Fanuc TP program (LS listing): ground_truth.ls

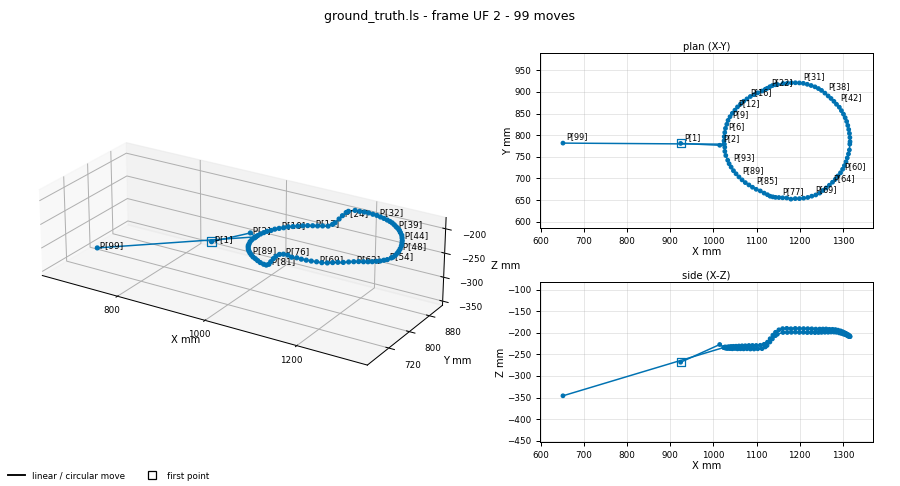
[picture p0: tool path of ground_truth.ls in frame UF 2, 99 of 99 moves have a stored position in this frame; points joined in program order, loops and branches not executed]
/PROG  TOR_XL_LEARN_V10
/ATTR
OWNER		= MNEDITOR;
COMMENT		= "WeldPRO Auto-Gen";
PROG_SIZE	= 7125;
CREATE		= DATE 26-07-31  TIME 15:22:18;
MODIFIED	= DATE 26-07-31  TIME 15:55:46;
FILE_NAME	= TOR_XL_L;
VERSION		= 0;
LINE_COUNT	= 113;
MEMORY_SIZE	= 7445;
PROTECT		= READ_WRITE;
TCD:  STACK_SIZE	= 0,
      TASK_PRIORITY	= 50,
      TIME_SLICE	= 0,
      BUSY_LAMP_OFF	= 0,
      ABORT_REQUEST	= 0,
      PAUSE_REQUEST	= 0;
DEFAULT_GROUP	= 1,*,*,*,*;
CONTROL_CODE	= 00000000 00000000;
/APPL
/MN
   1:  !WeldPRO Auto-Generated TPP ;
   2:  !TOR_XL_2026, TOR_xl_2907 ;
   3:   ;
   4:  UFRAME_NUM=2 ;
   5:  UTOOL_NUM=2 ;
   6:  !Feature Approach ;
   7:J P[1] 100% FINE    ;
   8:   ;
   9:  !Segment1 ;
  10:L P[2] 2000mm/sec FINE    ;
  11:   ;
  12:  CALL LASER_OFF    ;
  13:L P[3] R[23:moving]mm/sec CNT100    ;
  14:L P[4] R[23:moving]mm/sec CNT100    ;
  15:L P[5] R[23:moving]mm/sec CNT100    ;
  16:L P[6] R[23:moving]mm/sec CNT100    ;
  17:L P[7] R[23:moving]mm/sec CNT100    ;
  18:L P[8] R[23:moving]mm/sec CNT100    ;
  19:L P[9] R[23:moving]mm/sec CNT100    ;
  20:L P[10] R[23:moving]mm/sec CNT100    ;
  21:L P[11] R[23:moving]mm/sec CNT100    ;
  22:L P[12] R[23:moving]mm/sec CNT100    ;
  23:L P[13] R[23:moving]mm/sec CNT100    ;
  24:L P[14] R[23:moving]mm/sec CNT100    ;
  25:L P[15] R[23:moving]mm/sec CNT100    ;
  26:L P[16] R[23:moving]mm/sec CNT100    ;
  27:L P[17] R[23:moving]mm/sec CNT100    ;
  28:L P[18] R[23:moving]mm/sec CNT100    ;
  29:L P[19] R[23:moving]mm/sec CNT100    ;
  30:L P[20] R[23:moving]mm/sec CNT100    ;
  31:L P[21] R[23:moving]mm/sec CNT100    ;
  32:L P[22] R[23:moving]mm/sec CNT100    ;
  33:L P[23] R[23:moving]mm/sec CNT100    ;
  34:L P[24] R[23:moving]mm/sec CNT100    ;
  35:L P[25] R[23:moving]mm/sec CNT100    ;
  36:L P[26] R[23:moving]mm/sec CNT100    ;
  37:L P[27] R[23:moving]mm/sec CNT100    ;
  38:L P[28] R[23:moving]mm/sec CNT100    ;
  39:L P[29] R[23:moving]mm/sec CNT100    ;
  40:L P[30] R[23:moving]mm/sec CNT100    ;
  41:L P[31] R[23:moving]mm/sec CNT100    ;
  42:L P[32] R[23:moving]mm/sec CNT100    ;
  43:L P[33] R[23:moving]mm/sec CNT100    ;
  44:L P[34] R[23:moving]mm/sec CNT100    ;
  45:L P[35] R[23:moving]mm/sec CNT100    ;
  46:L P[36] R[23:moving]mm/sec CNT100    ;
  47:L P[37] R[23:moving]mm/sec CNT100    ;
  48:L P[38] R[23:moving]mm/sec CNT100    ;
  49:L P[39] R[23:moving]mm/sec CNT100    ;
  50:L P[40] R[23:moving]mm/sec CNT100    ;
  51:L P[41] R[23:moving]mm/sec CNT100    ;
  52:L P[42] R[23:moving]mm/sec CNT100    ;
  53:L P[43] R[23:moving]mm/sec CNT100    ;
  54:L P[44] R[23:moving]mm/sec CNT100    ;
  55:L P[45] R[23:moving]mm/sec CNT100    ;
  56:L P[46] R[23:moving]mm/sec CNT100    ;
  57:L P[47] R[23:moving]mm/sec CNT100    ;
  58:L P[48] R[23:moving]mm/sec CNT100    ;
  59:L P[49] R[23:moving]mm/sec CNT100    ;
  60:L P[50] R[23:moving]mm/sec CNT100    ;
  61:L P[51] R[23:moving]mm/sec CNT100    ;
  62:L P[52] R[23:moving]mm/sec CNT100    ;
  63:L P[53] R[23:moving]mm/sec CNT100    ;
  64:L P[54] R[23:moving]mm/sec CNT100    ;
  65:L P[55] R[23:moving]mm/sec CNT100    ;
  66:L P[56] R[23:moving]mm/sec CNT100    ;
  67:L P[57] R[23:moving]mm/sec CNT100    ;
  68:L P[58] R[23:moving]mm/sec CNT100    ;
  69:L P[59] R[23:moving]mm/sec CNT100    ;
  70:L P[60] R[23:moving]mm/sec CNT100    ;
  71:L P[61] R[23:moving]mm/sec CNT100    ;
  72:L P[62] R[23:moving]mm/sec CNT100    ;
  73:L P[63] R[23:moving]mm/sec CNT100    ;
  74:L P[64] R[23:moving]mm/sec CNT100    ;
  75:L P[65] R[23:moving]mm/sec CNT100    ;
  76:L P[66] R[23:moving]mm/sec CNT100    ;
  77:L P[67] R[23:moving]mm/sec CNT100    ;
  78:L P[68] R[23:moving]mm/sec CNT100    ;
  79:L P[69] R[23:moving]mm/sec CNT100    ;
  80:L P[70] R[23:moving]mm/sec CNT100    ;
  81:L P[71] R[23:moving]mm/sec CNT100    ;
  82:L P[72] R[23:moving]mm/sec CNT100    ;
  83:L P[73] R[23:moving]mm/sec CNT100    ;
  84:L P[74] R[23:moving]mm/sec CNT100    ;
  85:L P[75] R[23:moving]mm/sec CNT100    ;
  86:L P[76] R[23:moving]mm/sec CNT100    ;
  87:L P[77] R[23:moving]mm/sec CNT100    ;
  88:L P[78] R[23:moving]mm/sec CNT100    ;
  89:L P[79] R[23:moving]mm/sec CNT100    ;
  90:L P[80] R[23:moving]mm/sec CNT100    ;
  91:L P[81] R[23:moving]mm/sec CNT100    ;
  92:L P[82] R[23:moving]mm/sec CNT100    ;
  93:L P[83] R[23:moving]mm/sec CNT100    ;
  94:L P[84] R[23:moving]mm/sec CNT100    ;
  95:L P[85] R[23:moving]mm/sec CNT100    ;
  96:L P[86] R[23:moving]mm/sec CNT100    ;
  97:L P[87] R[23:moving]mm/sec CNT100    ;
  98:L P[88] R[23:moving]mm/sec CNT100    ;
  99:L P[89] R[23:moving]mm/sec CNT100    ;
 100:L P[90] R[23:moving]mm/sec CNT100    ;
 101:L P[91] R[23:moving]mm/sec CNT100    ;
 102:L P[92] R[23:moving]mm/sec CNT100    ;
 103:L P[93] R[23:moving]mm/sec CNT100    ;
 104:L P[94] R[23:moving]mm/sec CNT100    ;
 105:L P[95] R[23:moving]mm/sec CNT100    ;
 106:L P[96] R[23:moving]mm/sec CNT100    ;
 107:L P[97] R[23:moving]mm/sec CNT100    ;
 108:L P[98] R[23:moving]mm/sec FINE    ;
 109:  CALL LASER_OFF    ;
 110:   ;
 111:  !Feature Retreat ;
 112:L P[99] 2000mm/sec FINE    ;
 113:  CALL ROTATE    ;
/POS
P[1]{
   GP1:
	UF : 2, UT : 2,		CONFIG : 'F D T, 0, 0, 0',
	X =   924.335  mm,	Y =   780.986  mm,	Z =  -268.284  mm,
	W =  -106.495 deg,	P =   -15.000 deg,	R =    94.234 deg
};
P[2]{
   GP1:
	UF : 2, UT : 2,		CONFIG : 'F D T, 0, 0, 0',
	X =  1014.789  mm,	Y =   776.665  mm,	Z =  -227.278  mm,
	W =  -106.497 deg,	P =   -14.995 deg,	R =    94.216 deg
};
P[3]{
   GP1:
	UF : 2, UT : 2,		CONFIG : 'F D T, 0, 0, 0',
	X =  1024.819  mm,	Y =   779.312  mm,	Z =  -234.214  mm,
	W =  -106.501 deg,	P =   -14.998 deg,	R =    94.232 deg
};
P[4]{
   GP1:
	UF : 2, UT : 2,		CONFIG : 'F D T, 0, 0, 0',
	X =  1024.807  mm,	Y =   787.035  mm,	Z =  -234.284  mm,
	W =  -106.497 deg,	P =   -15.098 deg,	R =    90.375 deg
};
P[5]{
   GP1:
	UF : 2, UT : 2,		CONFIG : 'F D T, 0, 0, 0',
	X =  1025.197  mm,	Y =   796.630  mm,	Z =  -234.431  mm,
	W =  -106.481 deg,	P =   -15.217 deg,	R =    85.597 deg
};
P[6]{
   GP1:
	UF : 2, UT : 2,		CONFIG : 'F D T, 0, 0, 0',
	X =  1026.459  mm,	Y =   806.252  mm,	Z =  -234.929  mm,
	W =  -106.456 deg,	P =   -15.334 deg,	R =    80.807 deg
};
P[7]{
   GP1:
	UF : 2, UT : 2,		CONFIG : 'F D T, 0, 0, 0',
	X =  1028.142  mm,	Y =   815.795  mm,	Z =  -235.323  mm,
	W =  -106.423 deg,	P =   -15.450 deg,	R =    76.083 deg
};
P[8]{
   GP1:
	UF : 2, UT : 2,		CONFIG : 'F D T, 0, 0, 0',
	X =  1031.142  mm,	Y =   825.143  mm,	Z =  -236.265  mm,
	W =  -106.379 deg,	P =   -15.565 deg,	R =    71.210 deg
};
P[9]{
   GP1:
	UF : 2, UT : 2,		CONFIG : 'F D T, 0, 0, 0',
	X =  1034.075  mm,	Y =   834.282  mm,	Z =  -236.286  mm,
	W =  -106.322 deg,	P =   -15.679 deg,	R =    66.207 deg
};
P[10]{
   GP1:
	UF : 2, UT : 2,		CONFIG : 'F D T, 0, 0, 0',
	X =  1038.673  mm,	Y =   842.768  mm,	Z =  -236.720  mm,
	W =  -106.254 deg,	P =   -15.791 deg,	R =    61.015 deg
};
P[11]{
   GP1:
	UF : 2, UT : 2,		CONFIG : 'F D T, 0, 0, 0',
	X =  1044.018  mm,	Y =   850.684  mm,	Z =  -237.130  mm,
	W =  -106.180 deg,	P =   -15.896 deg,	R =    55.976 deg
};
P[12]{
   GP1:
	UF : 2, UT : 2,		CONFIG : 'F D T, 0, 0, 0',
	X =  1049.984  mm,	Y =   857.894  mm,	Z =  -236.475  mm,
	W =  -106.096 deg,	P =   -15.986 deg,	R =    51.162 deg
};
P[13]{
   GP1:
	UF : 2, UT : 2,		CONFIG : 'F D T, 0, 0, 0',
	X =  1055.988  mm,	Y =   865.483  mm,	Z =  -237.302  mm,
	W =  -106.012 deg,	P =   -16.067 deg,	R =    46.628 deg
};
P[14]{
   GP1:
	UF : 2, UT : 2,		CONFIG : 'F D T, 0, 0, 0',
	X =  1062.915  mm,	Y =   871.946  mm,	Z =  -237.205  mm,
	W =  -105.919 deg,	P =   -16.142 deg,	R =    41.952 deg
};
P[15]{
   GP1:
	UF : 2, UT : 2,		CONFIG : 'F D T, 0, 0, 0',
	X =  1070.115  mm,	Y =   878.600  mm,	Z =  -237.364  mm,
	W =  -105.870 deg,	P =   -16.177 deg,	R =    39.609 deg
};
P[16]{
   GP1:
	UF : 2, UT : 2,		CONFIG : 'F D T, 0, 0, 0',
	X =  1077.825  mm,	Y =   884.048  mm,	Z =  -237.128  mm,
	W =  -105.777 deg,	P =   -16.235 deg,	R =    35.365 deg
};
P[17]{
   GP1:
	UF : 2, UT : 2,		CONFIG : 'F D T, 0, 0, 0',
	X =  1085.741  mm,	Y =   889.534  mm,	Z =  -237.642  mm,
	W =  -105.677 deg,	P =   -16.289 deg,	R =    30.964 deg
};
P[18]{
   GP1:
	UF : 2, UT : 2,		CONFIG : 'F D T, 0, 0, 0',
	X =  1094.256  mm,	Y =   893.782  mm,	Z =  -237.649  mm,
	W =  -105.579 deg,	P =   -16.333 deg,	R =    26.830 deg
};
P[19]{
   GP1:
	UF : 2, UT : 2,		CONFIG : 'F D T, 0, 0, 0',
	X =  1102.826  mm,	Y =   898.014  mm,	Z =  -237.175  mm,
	W =  -105.535 deg,	P =   -16.344 deg,	R =    25.007 deg
};
P[20]{
   GP1:
	UF : 2, UT : 2,		CONFIG : 'F D T, 0, 0, 0',
	X =  1112.677  mm,	Y =   902.287  mm,	Z =  -236.848  mm,
	W =  -116.027 deg,	P =   -16.063 deg,	R =    30.267 deg
};
P[21]{
   GP1:
	UF : 2, UT : 2,		CONFIG : 'F D T, 0, 0, 0',
	X =  1120.220  mm,	Y =   906.262  mm,	Z =  -232.858  mm,
	W =  -126.877 deg,	P =   -15.356 deg,	R =    25.893 deg
};
P[22]{
   GP1:
	UF : 2, UT : 2,		CONFIG : 'F D T, 0, 0, 0',
	X =  1124.394  mm,	Y =   908.354  mm,	Z =  -229.385  mm,
	W =  -121.184 deg,	P =   -15.973 deg,	R =    18.444 deg
};
P[23]{
   GP1:
	UF : 2, UT : 2,		CONFIG : 'F D T, 0, 0, 0',
	X =  1130.913  mm,	Y =   912.231  mm,	Z =  -221.471  mm,
	W =  -115.329 deg,	P =   -16.208 deg,	R =    11.788 deg
};
P[24]{
   GP1:
	UF : 2, UT : 2,		CONFIG : 'F D T, 0, 0, 0',
	X =  1136.659  mm,	Y =   914.820  mm,	Z =  -214.206  mm,
	W =  -112.639 deg,	P =   -16.315 deg,	R =     9.714 deg
};
P[25]{
   GP1:
	UF : 2, UT : 2,		CONFIG : 'F D T, 0, 0, 0',
	X =  1143.585  mm,	Y =   916.753  mm,	Z =  -206.769  mm,
	W =  -110.015 deg,	P =   -16.386 deg,	R =     9.649 deg
};
P[26]{
   GP1:
	UF : 2, UT : 2,		CONFIG : 'F D T, 0, 0, 0',
	X =  1148.127  mm,	Y =   917.333  mm,	Z =  -203.429  mm,
	W =  -108.552 deg,	P =   -16.418 deg,	R =     8.950 deg
};
P[27]{
   GP1:
	UF : 2, UT : 2,		CONFIG : 'F D T, 0, 0, 0',
	X =  1161.287  mm,	Y =   919.693  mm,	Z =  -199.396  mm,
	W =  -105.409 deg,	P =   -16.443 deg,	R =     6.805 deg
};
P[28]{
   GP1:
	UF : 2, UT : 2,		CONFIG : 'F D T, 0, 0, 0',
	X =  1171.157  mm,	Y =   920.269  mm,	Z =  -199.402  mm,
	W =  -104.866 deg,	P =   -16.444 deg,	R =     5.597 deg
};
P[29]{
   GP1:
	UF : 2, UT : 2,		CONFIG : 'F D T, 0, 0, 0',
	X =  1180.649  mm,	Y =   921.254  mm,	Z =  -199.064  mm,
	W =  -104.887 deg,	P =   -16.444 deg,	R =     3.523 deg
};
P[30]{
   GP1:
	UF : 2, UT : 2,		CONFIG : 'F D T, 0, 0, 0',
	X =  1189.853  mm,	Y =   921.397  mm,	Z =  -198.761  mm,
	W =  -104.930 deg,	P =   -16.439 deg,	R =     -.729 deg
};
P[31]{
   GP1:
	UF : 2, UT : 2,		CONFIG : 'F D T, 0, 0, 0',
	X =  1199.182  mm,	Y =   920.957  mm,	Z =  -199.232  mm,
	W =  -104.979 deg,	P =   -16.424 deg,	R =    -5.541 deg
};
P[32]{
   GP1:
	UF : 2, UT : 2,		CONFIG : 'F D T, 0, 0, 0',
	X =  1208.351  mm,	Y =   920.022  mm,	Z =  -199.133  mm,
	W =  -105.028 deg,	P =   -16.400 deg,	R =   -10.259 deg
};
P[33]{
   GP1:
	UF : 2, UT : 2,		CONFIG : 'F D T, 0, 0, 0',
	X =  1217.485  mm,	Y =   917.761  mm,	Z =  -199.566  mm,
	W =  -105.070 deg,	P =   -16.371 deg,	R =   -14.490 deg
};
P[34]{
   GP1:
	UF : 2, UT : 2,		CONFIG : 'F D T, 0, 0, 0',
	X =  1226.426  mm,	Y =   915.001  mm,	Z =  -199.462  mm,
	W =  -105.112 deg,	P =   -16.334 deg,	R =   -18.515 deg
};
P[35]{
   GP1:
	UF : 2, UT : 2,		CONFIG : 'F D T, 0, 0, 0',
	X =  1235.239  mm,	Y =   911.936  mm,	Z =  -199.665  mm,
	W =  -105.158 deg,	P =   -16.285 deg,	R =   -23.051 deg
};
P[36]{
   GP1:
	UF : 2, UT : 2,		CONFIG : 'F D T, 0, 0, 0',
	X =  1243.244  mm,	Y =   907.972  mm,	Z =  -199.458  mm,
	W =  -105.219 deg,	P =   -16.204 deg,	R =   -29.417 deg
};
P[37]{
   GP1:
	UF : 2, UT : 2,		CONFIG : 'F D T, 0, 0, 0',
	X =  1250.416  mm,	Y =   903.609  mm,	Z =  -199.147  mm,
	W =  -105.311 deg,	P =   -16.047 deg,	R =   -39.415 deg
};
P[38]{
   GP1:
	UF : 2, UT : 2,		CONFIG : 'F D T, 0, 0, 0',
	X =  1258.217  mm,	Y =   897.390  mm,	Z =  -198.941  mm,
	W =  -105.307 deg,	P =   -16.055 deg,	R =   -38.974 deg
};
P[39]{
   GP1:
	UF : 2, UT : 2,		CONFIG : 'F D T, 0, 0, 0',
	X =  1265.775  mm,	Y =   890.850  mm,	Z =  -198.923  mm,
	W =  -105.302 deg,	P =   -16.063 deg,	R =   -38.625 deg
};
P[40]{
   GP1:
	UF : 2, UT : 2,		CONFIG : 'F D T, 0, 0, 0',
	X =  1272.442  mm,	Y =   885.004  mm,	Z =  -198.403  mm,
	W =  -105.469 deg,	P =   -15.944 deg,	R =   -44.977 deg
};
P[41]{
   GP1:
	UF : 2, UT : 2,		CONFIG : 'F D T, 0, 0, 0',
	X =  1279.129  mm,	Y =   878.386  mm,	Z =  -198.494  mm,
	W =  -105.661 deg,	P =   -15.890 deg,	R =   -47.714 deg
};
P[42]{
   GP1:
	UF : 2, UT : 2,		CONFIG : 'F D T, 0, 0, 0',
	X =  1285.054  mm,	Y =   871.499  mm,	Z =  -198.979  mm,
	W =  -106.210 deg,	P =   -15.792 deg,	R =   -52.259 deg
};
P[43]{
   GP1:
	UF : 2, UT : 2,		CONFIG : 'F D T, 0, 0, 0',
	X =  1291.590  mm,	Y =   864.741  mm,	Z =  -200.433  mm,
	W =  -106.927 deg,	P =   -15.688 deg,	R =   -56.663 deg
};
P[44]{
   GP1:
	UF : 2, UT : 2,		CONFIG : 'F D T, 0, 0, 0',
	X =  1296.495  mm,	Y =   856.855  mm,	Z =  -201.631  mm,
	W =  -107.603 deg,	P =   -15.597 deg,	R =   -60.244 deg
};
P[45]{
   GP1:
	UF : 2, UT : 2,		CONFIG : 'F D T, 0, 0, 0',
	X =  1301.221  mm,	Y =   848.739  mm,	Z =  -203.247  mm,
	W =  -108.271 deg,	P =   -15.504 deg,	R =   -63.686 deg
};
P[46]{
   GP1:
	UF : 2, UT : 2,		CONFIG : 'F D T, 0, 0, 0',
	X =  1305.143  mm,	Y =   840.488  mm,	Z =  -204.302  mm,
	W =  -109.143 deg,	P =   -15.378 deg,	R =   -68.203 deg
};
P[47]{
   GP1:
	UF : 2, UT : 2,		CONFIG : 'F D T, 0, 0, 0',
	X =  1308.602  mm,	Y =   831.819  mm,	Z =  -205.714  mm,
	W =  -109.899 deg,	P =   -15.253 deg,	R =   -72.505 deg
};
P[48]{
   GP1:
	UF : 2, UT : 2,		CONFIG : 'F D T, 0, 0, 0',
	X =  1311.203  mm,	Y =   822.479  mm,	Z =  -207.429  mm,
	W =  -110.273 deg,	P =   -15.181 deg,	R =   -74.982 deg
};
P[49]{
   GP1:
	UF : 2, UT : 2,		CONFIG : 'F D T, 0, 0, 0',
	X =  1313.345  mm,	Y =   813.167  mm,	Z =  -208.220  mm,
	W =  -110.634 deg,	P =   -14.305 deg,	R =   -78.233 deg
};
P[50]{
   GP1:
	UF : 2, UT : 2,		CONFIG : 'F D T, 0, 0, 0',
	X =  1315.073  mm,	Y =   804.056  mm,	Z =  -208.497  mm,
	W =  -111.054 deg,	P =   -14.769 deg,	R =   -83.165 deg
};
P[51]{
   GP1:
	UF : 2, UT : 2,		CONFIG : 'F D T, 0, 0, 0',
	X =  1316.073  mm,	Y =   794.665  mm,	Z =  -208.886  mm,
	W =  -111.189 deg,	P =   -15.306 deg,	R =   -88.309 deg
};
P[52]{
   GP1:
	UF : 2, UT : 2,		CONFIG : 'F D T, 0, 0, 0',
	X =  1316.411  mm,	Y =   785.001  mm,	Z =  -208.750  mm,
	W =  -111.129 deg,	P =   -15.645 deg,	R =   -91.614 deg
};
P[53]{
   GP1:
	UF : 2, UT : 2,		CONFIG : 'F D T, 0, 0, 0',
	X =  1315.842  mm,	Y =   779.373  mm,	Z =  -208.294  mm,
	W =  -110.924 deg,	P =   -15.048 deg,	R =   -94.524 deg
};
P[54]{
   GP1:
	UF : 2, UT : 2,		CONFIG : 'F D T, 0, 0, 0',
	X =  1314.913  mm,	Y =   765.868  mm,	Z =  -206.750  mm,
	W =  -110.275 deg,	P =   -14.535 deg,	R =  -100.837 deg
};
P[55]{
   GP1:
	UF : 2, UT : 2,		CONFIG : 'F D T, 0, 0, 0',
	X =  1312.784  mm,	Y =   756.634  mm,	Z =  -204.950  mm,
	W =  -109.632 deg,	P =   -14.447 deg,	R =  -105.266 deg
};
P[56]{
   GP1:
	UF : 2, UT : 2,		CONFIG : 'F D T, 0, 0, 0',
	X =  1310.011  mm,	Y =   747.385  mm,	Z =  -203.665  mm,
	W =  -109.082 deg,	P =   -14.382 deg,	R =  -108.626 deg
};
P[57]{
   GP1:
	UF : 2, UT : 2,		CONFIG : 'F D T, 0, 0, 0',
	X =  1307.077  mm,	Y =   738.446  mm,	Z =  -201.496  mm,
	W =  -108.349 deg,	P =   -14.302 deg,	R =  -112.873 deg
};
P[58]{
   GP1:
	UF : 2, UT : 2,		CONFIG : 'F D T, 0, 0, 0',
	X =  1303.385  mm,	Y =   729.562  mm,	Z =  -199.729  mm,
	W =  -107.748 deg,	P =   -14.239 deg,	R =  -116.265 deg
};
P[59]{
   GP1:
	UF : 2, UT : 2,		CONFIG : 'F D T, 0, 0, 0',
	X =  1299.269  mm,	Y =   721.118  mm,	Z =  -197.625  mm,
	W =  -106.924 deg,	P =   -14.148 deg,	R =  -121.192 deg
};
P[60]{
   GP1:
	UF : 2, UT : 2,		CONFIG : 'F D T, 0, 0, 0',
	X =  1294.374  mm,	Y =   713.041  mm,	Z =  -195.656  mm,
	W =  -106.269 deg,	P =   -14.066 deg,	R =  -125.698 deg
};
P[61]{
   GP1:
	UF : 2, UT : 2,		CONFIG : 'F D T, 0, 0, 0',
	X =  1288.358  mm,	Y =   705.703  mm,	Z =  -194.002  mm,
	W =  -105.781 deg,	P =   -13.988 deg,	R =  -130.143 deg
};
P[62]{
   GP1:
	UF : 2, UT : 2,		CONFIG : 'F D T, 0, 0, 0',
	X =  1282.492  mm,	Y =   698.100  mm,	Z =  -192.726  mm,
	W =  -105.526 deg,	P =   -13.913 deg,	R =  -134.519 deg
};
P[63]{
   GP1:
	UF : 2, UT : 2,		CONFIG : 'F D T, 0, 0, 0',
	X =  1275.865  mm,	Y =   691.153  mm,	Z =  -192.125  mm,
	W =  -105.437 deg,	P =   -13.849 deg,	R =  -138.629 deg
};
P[64]{
   GP1:
	UF : 2, UT : 2,		CONFIG : 'F D T, 0, 0, 0',
	X =  1268.646  mm,	Y =   684.300  mm,	Z =  -192.114  mm,
	W =  -105.429 deg,	P =   -13.831 deg,	R =  -139.837 deg
};
P[65]{
   GP1:
	UF : 2, UT : 2,		CONFIG : 'F D T, 0, 0, 0',
	X =  1261.055  mm,	Y =   677.915  mm,	Z =  -191.269  mm,
	W =  -105.443 deg,	P =   -13.863 deg,	R =  -137.727 deg
};
P[66]{
   GP1:
	UF : 2, UT : 2,		CONFIG : 'F D T, 0, 0, 0',
	X =  1253.614  mm,	Y =   672.078  mm,	Z =  -191.403  mm,
	W =  -105.373 deg,	P =   -13.729 deg,	R =  -147.436 deg
};
P[67]{
   GP1:
	UF : 2, UT : 2,		CONFIG : 'F D T, 0, 0, 0',
	X =  1246.068  mm,	Y =   665.962  mm,	Z =  -191.505  mm,
	W =  -105.298 deg,	P =   -13.637 deg,	R =  -156.529 deg
};
P[68]{
   GP1:
	UF : 2, UT : 2,		CONFIG : 'F D T, 0, 0, 0',
	X =  1237.101  mm,	Y =   661.714  mm,	Z =  -191.526  mm,
	W =  -105.277 deg,	P =   -13.618 deg,	R =  -158.977 deg
};
P[69]{
   GP1:
	UF : 2, UT : 2,		CONFIG : 'F D T, 0, 0, 0',
	X =  1227.843  mm,	Y =   658.867  mm,	Z =  -190.889  mm,
	W =  -105.241 deg,	P =   -13.592 deg,	R =  -162.969 deg
};
P[70]{
   GP1:
	UF : 2, UT : 2,		CONFIG : 'F D T, 0, 0, 0',
	X =  1218.505  mm,	Y =   655.896  mm,	Z =  -190.592  mm,
	W =  -105.201 deg,	P =   -13.569 deg,	R =  -167.030 deg
};
P[71]{
   GP1:
	UF : 2, UT : 2,		CONFIG : 'F D T, 0, 0, 0',
	X =  1208.933  mm,	Y =   654.240  mm,	Z =  -190.461  mm,
	W =  -105.159 deg,	P =   -13.560 deg,	R =  -171.569 deg
};
P[72]{
   GP1:
	UF : 2, UT : 2,		CONFIG : 'F D T, 0, 0, 0',
	X =  1199.274  mm,	Y =   653.204  mm,	Z =  -190.365  mm,
	W =  -105.113 deg,	P =   -13.556 deg,	R =  -176.312 deg
};
P[73]{
   GP1:
	UF : 2, UT : 2,		CONFIG : 'F D T, 0, 0, 0',
	X =  1189.625  mm,	Y =   653.291  mm,	Z =  -190.022  mm,
	W =  -105.068 deg,	P =   -13.561 deg,	R =   179.213 deg
};
P[74]{
   GP1:
	UF : 2, UT : 2,		CONFIG : 'F D T, 0, 0, 0',
	X =  1179.533  mm,	Y =   652.020  mm,	Z =  -190.760  mm,
	W =  -105.038 deg,	P =   -13.569 deg,	R =   176.231 deg
};
P[75]{
   GP1:
	UF : 2, UT : 2,		CONFIG : 'F D T, 0, 0, 0',
	X =  1169.974  mm,	Y =   654.662  mm,	Z =  -189.842  mm,
	W =  -105.207 deg,	P =   -13.572 deg,	R =   175.290 deg
};
P[76]{
   GP1:
	UF : 2, UT : 2,		CONFIG : 'F D T, 0, 0, 0',
	X =  1160.471  mm,	Y =   655.101  mm,	Z =  -190.495  mm,
	W =  -107.012 deg,	P =   -13.569 deg,	R =   174.537 deg
};
P[77]{
   GP1:
	UF : 2, UT : 2,		CONFIG : 'F D T, 0, 0, 0',
	X =  1151.749  mm,	Y =   655.749  mm,	Z =  -193.260  mm,
	W =  -109.414 deg,	P =   -13.538 deg,	R =   174.483 deg
};
P[78]{
   GP1:
	UF : 2, UT : 2,		CONFIG : 'F D T, 0, 0, 0',
	X =  1143.955  mm,	Y =   656.114  mm,	Z =  -199.016  mm,
	W =  -112.196 deg,	P =   -13.466 deg,	R =   175.322 deg
};
P[79]{
   GP1:
	UF : 2, UT : 2,		CONFIG : 'F D T, 0, 0, 0',
	X =  1137.830  mm,	Y =   657.303  mm,	Z =  -205.654  mm,
	W =  -114.872 deg,	P =   -13.369 deg,	R =   175.421 deg
};
P[80]{
   GP1:
	UF : 2, UT : 2,		CONFIG : 'F D T, 0, 0, 0',
	X =  1131.505  mm,	Y =   658.719  mm,	Z =  -213.846  mm,
	W =  -120.114 deg,	P =   -13.109 deg,	R =   172.292 deg
};
P[81]{
   GP1:
	UF : 2, UT : 2,		CONFIG : 'F D T, 0, 0, 0',
	X =  1125.289  mm,	Y =   662.259  mm,	Z =  -221.845  mm,
	W =  -126.807 deg,	P =   -12.619 deg,	R =   167.802 deg
};
P[82]{
   GP1:
	UF : 2, UT : 2,		CONFIG : 'F D T, 0, 0, 0',
	X =  1117.564  mm,	Y =   665.974  mm,	Z =  -226.761  mm,
	W =  -119.561 deg,	P =   -13.285 deg,	R =   157.805 deg
};
P[83]{
   GP1:
	UF : 2, UT : 2,		CONFIG : 'F D T, 0, 0, 0',
	X =  1108.729  mm,	Y =   670.990  mm,	Z =  -229.075  mm,
	W =  -107.325 deg,	P =   -13.741 deg,	R =   154.436 deg
};
P[84]{
   GP1:
	UF : 2, UT : 2,		CONFIG : 'F D T, 0, 0, 0',
	X =  1099.274  mm,	Y =   674.765  mm,	Z =  -229.504  mm,
	W =  -105.746 deg,	P =   -13.749 deg,	R =   154.142 deg
};
P[85]{
   GP1:
	UF : 2, UT : 2,		CONFIG : 'F D T, 0, 0, 0',
	X =  1090.619  mm,	Y =   679.528  mm,	Z =  -229.465  mm,
	W =  -105.804 deg,	P =   -13.784 deg,	R =   151.505 deg
};
P[86]{
   GP1:
	UF : 2, UT : 2,		CONFIG : 'F D T, 0, 0, 0',
	X =  1082.353  mm,	Y =   684.900  mm,	Z =  -229.555  mm,
	W =  -105.885 deg,	P =   -13.838 deg,	R =   147.738 deg
};
P[87]{
   GP1:
	UF : 2, UT : 2,		CONFIG : 'F D T, 0, 0, 0',
	X =  1074.034  mm,	Y =   690.284  mm,	Z =  -230.136  mm,
	W =  -105.988 deg,	P =   -13.918 deg,	R =   142.681 deg
};
P[88]{
   GP1:
	UF : 2, UT : 2,		CONFIG : 'F D T, 0, 0, 0',
	X =  1066.503  mm,	Y =   696.595  mm,	Z =  -230.271  mm,
	W =  -106.084 deg,	P =   -14.001 deg,	R =   137.677 deg
};
P[89]{
   GP1:
	UF : 2, UT : 2,		CONFIG : 'F D T, 0, 0, 0',
	X =  1059.343  mm,	Y =   703.420  mm,	Z =  -230.710  mm,
	W =  -106.129 deg,	P =   -14.056 deg,	R =   135.014 deg
};
P[90]{
   GP1:
	UF : 2, UT : 2,		CONFIG : 'F D T, 0, 0, 0',
	X =  1052.586  mm,	Y =   710.718  mm,	Z =  -231.224  mm,
	W =  -106.186 deg,	P =   -14.117 deg,	R =   131.621 deg
};
P[91]{
   GP1:
	UF : 2, UT : 2,		CONFIG : 'F D T, 0, 0, 0',
	X =  1046.607  mm,	Y =   717.883  mm,	Z =  -231.451  mm,
	W =  -106.269 deg,	P =   -14.234 deg,	R =   126.207 deg
};
P[92]{
   GP1:
	UF : 2, UT : 2,		CONFIG : 'F D T, 0, 0, 0',
	X =  1041.207  mm,	Y =   726.172  mm,	Z =  -231.735  mm,
	W =  -106.343 deg,	P =   -14.367 deg,	R =   120.225 deg
};
P[93]{
   GP1:
	UF : 2, UT : 2,		CONFIG : 'F D T, 0, 0, 0',
	X =  1036.574  mm,	Y =   733.935  mm,	Z =  -232.344  mm,
	W =  -106.383 deg,	P =   -14.448 deg,	R =   116.672 deg
};
P[94]{
   GP1:
	UF : 2, UT : 2,		CONFIG : 'F D T, 0, 0, 0',
	X =  1033.279  mm,	Y =   742.080  mm,	Z =  -232.849  mm,
	W =  -106.433 deg,	P =   -14.556 deg,	R =   111.957 deg
};
P[95]{
   GP1:
	UF : 2, UT : 2,		CONFIG : 'F D T, 0, 0, 0',
	X =  1028.866  mm,	Y =   752.999  mm,	Z =  -233.214  mm,
	W =  -106.465 deg,	P =   -14.714 deg,	R =   105.666 deg
};
P[96]{
   GP1:
	UF : 2, UT : 2,		CONFIG : 'F D T, 0, 1, 0',
	X =  1026.636  mm,	Y =   762.583  mm,	Z =  -233.481  mm,
	W =  -106.480 deg,	P =   -14.798 deg,	R =   102.261 deg
};
P[97]{
   GP1:
	UF : 2, UT : 2,		CONFIG : 'F D T, 0, 1, 0',
	X =  1026.457  mm,	Y =   772.200  mm,	Z =  -233.294  mm,
	W =  -106.494 deg,	P =   -14.935 deg,	R =    96.827 deg
};
P[98]{
   GP1:
	UF : 2, UT : 2,		CONFIG : 'F D T, 0, 1, 0',
	X =  1025.303  mm,	Y =   779.231  mm,	Z =  -233.864  mm,
	W =  -106.501 deg,	P =   -15.000 deg,	R =    94.235 deg
};
P[99]{
   GP1:
	UF : 2, UT : 2,		CONFIG : 'F D T, 0, 1, 0',
	X =   651.995  mm,	Y =   781.694  mm,	Z =  -345.952  mm,
	W =  -106.495 deg,	P =   -15.000 deg,	R =    94.234 deg
};
/END
